{attribute addProperty BoxType "AX5160-0000-0210-0210"}
{attribute addProperty Id "AT_xAT %I*AT_x_15FCA3A680100MDTAT %Q*MDT_C2B17B7F4860WcStateAT %I*WcState_98A4DF7520.250InfoDataAT %I*InfoData_AEB17F4D152190"}
{attribute addProperty CRC "2773434183"}
{attribute addProperty SizeInBites "282"}
{attribute addProperty SizeInBytes "35.25"}
TYPE AX5160_3FB01CDA :
STRUCT
	{attribute addProperty Name "AT_x"}
	AT_x : AT_x_15FCA3A6;
	{attribute addProperty Name "MDT"}
	MDT : MDT_C2B17B7F;
	{attribute addProperty Name "WcState"}
	WcState : WcState_98A4DF75;
	{attribute addProperty Name "InfoData"}
	InfoData : InfoData_AEB17F4D;
END_STRUCT
END_TYPE

(* stored: Version 1.2.0.0, ProductVersion 3.1.4024.9
   DUT AX5160_3FB01CDA: Id {ad6d0656-cd91-4a8f-9678-bfada426aac4} *)
